FUNCTION_BLOCK Sensor (* Composite Function Block Type *)
  (* Standard: 61499-2 *)
  (* Version 0.0, 9/14/2008, Horst Mayer, nxtControl GmbH, template *)
  PACKAGE Main;
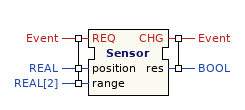
  EVENT_INPUT
    REQ WITH position, range; (* Normal Execution Request *)
  END_EVENT
  EVENT_OUTPUT
    CHG WITH res; (* Execution Confirmation *)
  END_EVENT
  VAR_INPUT
    position : REAL;
    range : ARRAY [0..1] OF REAL;
  END_VAR
  VAR_OUTPUT
    res : BOOL;
  END_VAR
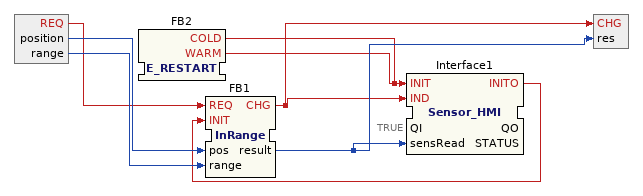
  FBS
    Interface1 : Sensor_HMI(QI := TRUE);
    FB1 : InRange;
    FB2 : E_RESTART;
  END_FBS
  EVENT_CONNECTIONS
    REQ TO FB1.REQ;
    FB1.CHG TO CHG;
    FB2.COLD TO Interface1.INIT;
    FB2.WARM TO Interface1.INIT;
    FB1.CHG TO Interface1.IND;
    Interface1.INITO TO FB1.INIT;
  END_CONNECTIONS
  DATA_CONNECTIONS
    FB1.result TO res;
    position TO FB1.pos;
    range TO FB1.range;
    FB1.result TO Interface1.sensRead;
  END_CONNECTIONS
END_FUNCTION_BLOCK
